Fanuc KAREL source: INI_DYN_DISP.kl

PROGRAM T
%NOLOCKGROUP
VAR
 v0 : INTEGER
 v1 : INTEGER
 v2 : STRING[40]
 v3 : INTEGER
 v4 : INTEGER
 v5 : INTEGER
 v6 : INTEGER
 v7 : INTEGER
 v8 : INTEGER
 v9 : ARRAY[10] OF STRING[40]
 v10 : INTEGER
BEGIN
 INI_DYN_DISP(v0, v1, v2, v3, v4, v5, v6, v7, v8, v9, v10)
END T
